INTERFACE ITF_SaMController

END_INTERFACE

(* stored: Version 1.1.0.1
   Itf ITF_SaMController: Id {c7f4a38b-e5fc-0e2c-38d0-203cc4e95405} *)
